Staubli VAL3: setSpeed.pgx

program setSpeed(string messageBuffer (dimensions=1), num sio_ID (dimensions=1))
  local num indexParam
  local bool isNumber
  local num numSpeedLoc
  local string reply
begin
  //**************************************************
  // Method to set the speed of the robot. Messages take the form:
  //     setSpeed:#20
  //**************************************************

  // Find the parameter in the stringMessage and convert to a number
  indexParam=find(messageBuffer,("#"))
  toNum(right(messageBuffer,(len(messageBuffer)-(indexParam+1))),numSpeedLoc,isNumber)

  // If conversion worked, set the speed; if not post a message and return
  if isNumber==false
    reply="setSpeed:fail_'Data is not a number'"
    putln(toString("",indexParam))
    putln(toString("",len(messageBuffer)-(indexParam+1)))
    put("Failed setting speed. Found: ")
    putln(right(messageBuffer,(len(messageBuffer)-indexParam)))
  else
    mFastMov.vel=numSpeedLoc
    put("Speed = ")
    putln(numSpeedLoc)
    reply="setSpeed:done"
  endIf

  taskCreate "sendStatus",10,sendStatus(reply,sio_ID)
end
